// TIA Portal V19 export
TYPE "TExtEncoder_Ctrl"
// stored: Access Published
   STRUCT
      Rst : Bool;   // Reset alarms
      Home : Bool;   // Home command
      HomeMode : Int;   // Home mode (see MC Home)
      HomePosition : LReal;   // Home position
   END_STRUCT;
END_TYPE
